// TwinCAT 3 PLC project PLC
// ProgramVersion: 3.1.4022.1
// libraries:
//   Tc2_Standard, * (Beckhoff Automation GmbH)
//   Tc2_System, * (Beckhoff Automation GmbH)
//   Tc3_Module, * (Beckhoff Automation GmbH)
//   VisuDialogs, * (System)
//   VisuSymbols,3.5.10.0,System
// project tree:
//   / GlobalTextList.TcGTLO, PlcTask.TcTTO, Visualization Manager.TcVMO (not stored)
//   POUs/ MAIN.TcPOU, POU.TcPOU
//   VISUs/ Visualization.TcVIS
// real-time tasks:
//   TASK PlcTask: cycle T#10ms, priority 20, ADS port 350

CONFIGURATION PLC
    RESOURCE PLC ON TwinCAT3
        TASK PlcTask(INTERVAL := T#10ms, PRIORITY := 20);
        PROGRAM MAIN WITH PlcTask : MAIN;
    END_RESOURCE
END_CONFIGURATION

// ---- POUs/MAIN.TcPOU
PROGRAM MAIN
VAR
END_VAR

POU();

END_PROGRAM

// ---- POUs/POU.TcPOU
PROGRAM POU
VAR
	up_inside: BOOL;
	door_up: BOOL;
	motor_up: BOOL;
	down_inside: BOOL;
	door_down: BOOL;
	motor_down: BOOL;
	motor_off: BOOL;
	key: BOOL;
	up_outside: BOOL;
	down_outside: BOOL;
	TON_0 : TON;
	TON0_et: TIME;
	TON_1: TON;	
	TON1_et: Time;
END_VAR
VAR // added by the converter: edge detectors and wires of the graphical bodies
    _w1, _w2, _w3, _w4, _w5, _w6 : BOOL;
END_VAR

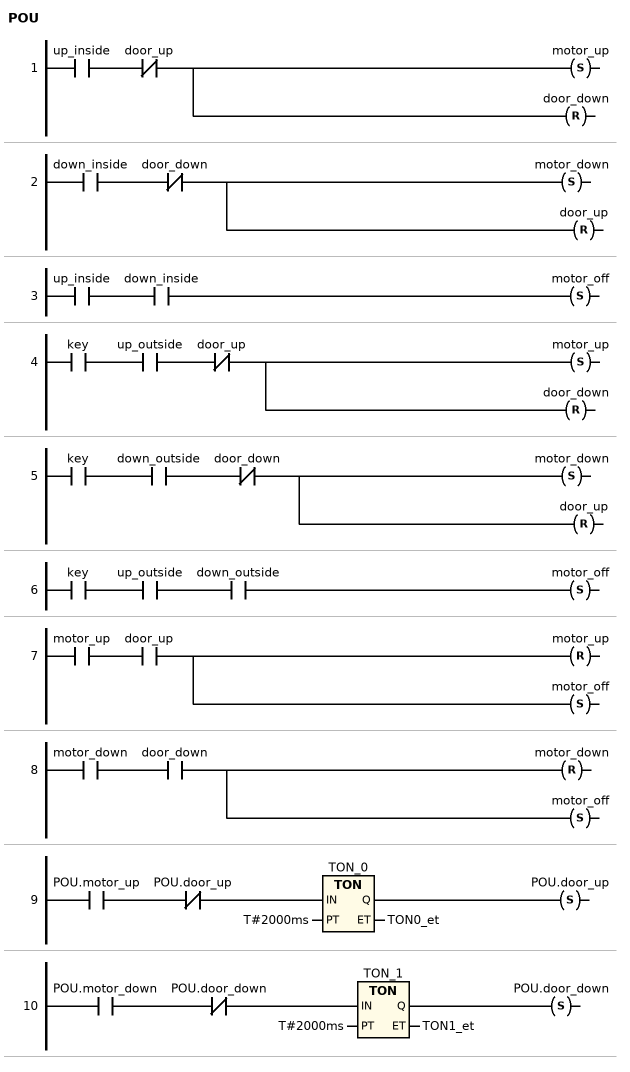
// NETWORK 1
_w1 := up_inside AND NOT door_up;
motor_up S= _w1;
door_down R= _w1;

// NETWORK 2
_w2 := down_inside AND NOT door_down;
motor_down S= _w2;
door_up R= _w2;

// NETWORK 3
motor_off S= up_inside AND down_inside;

// NETWORK 4
_w3 := key AND up_outside AND NOT door_up;
motor_up S= _w3;
door_down R= _w3;

// NETWORK 5
_w4 := key AND down_outside AND NOT door_down;
motor_down S= _w4;
door_up R= _w4;

// NETWORK 6
motor_off S= key AND up_outside AND down_outside;

// NETWORK 7
_w5 := motor_up AND door_up;
motor_up R= _w5;
motor_off S= _w5;

// NETWORK 8
_w6 := motor_down AND door_down;
motor_down R= _w6;
motor_off S= _w6;

// NETWORK 9
TON_0(IN := POU.motor_up AND NOT POU.door_up, PT := T#2000ms, ET => TON0_et); // TON
POU.door_up S= TON_0.Q;

// NETWORK 10
TON_1(IN := POU.motor_down AND NOT POU.door_down, PT := T#2000ms, ET => TON1_et); // TON
POU.door_down S= TON_1.Q;

END_PROGRAM

// ---- GlobalTextList.TcGTLO
TEXTLIST GlobalTextList
  217 = 'Door'
  286 = 'Down'
  402 = 'Garage Door Down'
  46 = 'Garage Door Up'
  367 = 'Inside'
  141 = 'Key'
  287 = 'Motor'
  877 = 'Motor Down'
  307 = 'Motor Up'
  797 = 'Outside'
  446 = 'Up'
  101 = 'Wee'
END_TEXTLIST

// ---- VISUs/Visualization.TcVIS
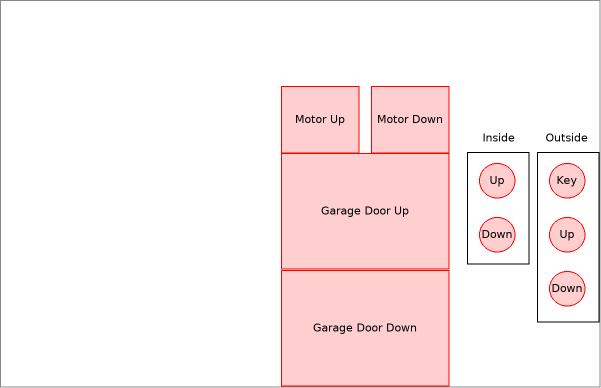
VISUALIZATION Visualization  // 601x388
    Rectangle (281,86 78x67), "Motor Up", colour toggle: POU.motor_up
    Rectangle (467,152 62x112)
    Rectangle (537,152 62x170)
    Ellipse (479,163 36x35), "Up", colour toggle: POU.up_inside
        OnMouseDown: toggle POU.up_inside
    Ellipse (549,163 36x35), "Key", colour toggle: POU.key
        OnMouseDown: toggle POU.key
    Ellipse (549,217 36x35), "Up", colour toggle: POU.up_outside
        OnMouseDown: toggle POU.up_outside
    Ellipse (549,271 36x35), "Down", colour toggle: POU.down_outside
        OnMouseDown: toggle POU.down_outside
    Ellipse (479,217 36x35), "Down", colour toggle: POU.down_inside
        OnMouseDown: toggle POU.down_inside
    Rectangle (281,153 168x116), "Garage Door Up", colour toggle: POU.door_up
        OnMouseDown: toggle POU.door_up
        OnMouseDown: toggle POU.door_up
    Rectangle (371,86 78x67), "Motor Down", colour toggle: POU.motor_down
    Rectangle (281,270 168x116), "Garage Door Down", colour toggle: POU.door_down
        OnMouseDown: toggle POU.door_down
    Label (474,123 50x30), "Inside"
    Label (542,123 50x30), "Outside"
END_VISUALIZATION
